(* PLC project  *)

PROGRAM P
  VAR  (* added by the conversion: wires and edge detectors of the diagram *)
    _ADD3_ENO : BOOL;
    _ADD3_OUT : ANY;
  END_VAR

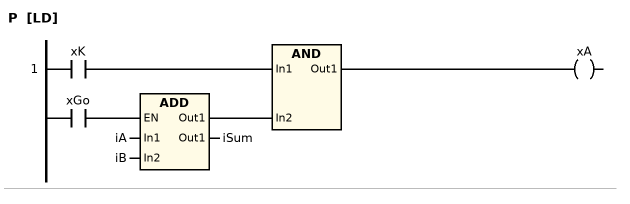
(* LD diagram, written out as Structured Text *)
_ADD3_OUT := ADD(EN := xGo, IN1 := iA, IN2 := iB, ENO => _ADD3_ENO);
xA := xK AND _ADD3_OUT;
IF _ADD3_ENO THEN iSum := _ADD3_OUT; END_IF;
END_PROGRAM
